// Mitsubishi GX Works2 project: LRI - PLC - A1+A2.A3   PLC: Q03UDV

PROGRAM MAIN
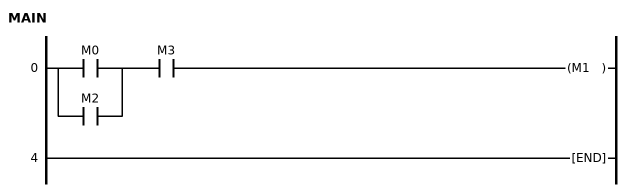
0     LD      M0
      OR      M2
      AND     M3
      OUT     M1
4     END
END_PROGRAM
